FUNCTION_BLOCK ABS_LINT (* IEC 61131-3,Table 23#1 *)
  (* Standard: 61131-3 *)
  (* Version 0.0, 2004-12-15, JHC, Rockwell Automation, Converted from SRC format. *)
  (* Compiler header: package fb.rt.plc.math; *)
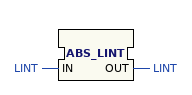
  VAR_INPUT
    IN : LINT;
  END_VAR
  VAR_OUTPUT
    OUT : LINT;
  END_VAR
END_FUNCTION_BLOCK
